FUNCTION_BLOCK FB_CalcThicknessFromXRayTransmission EXTENDS FB_Fallible IMPLEMENTS I_CalcThicknessFromXRayTransmission
VAR
    iConvertUnits : I_ConvertUnitsLREAL;
    iCalcXRayAbsorption : I_CalcXRayAbsorptionConstant;

    fbAbsorptionConstant : FB_QuantityLREALPublic(Units := '1/m');
    fbAbsorptionConstantum : FB_QuantityLREALPublic(Units := '1/um');
    fbThickness : FB_QuantityLREALPublic(Units := 'um');
END_VAR


METHOD Calculate
VAR_INPUT
    MaterialFormula : T_MaxString;
    Transmission : I_QuantityLREAL;
    Thickness : I_QuantityLREALPublic;
END_VAR

// Initialize error values
ClearError();

IF Transmission.GetError() THEN
    SetError(Msg :=
        CONCAT('Input transmission has an error: ',
        Transmission.GetErrorMsg())
    );
    Thickness.SetError(Msg := GetErrorMsg());
    RETURN;
END_IF

IF Transmission.Val <= 0.0 THEN
    SetError(Msg := 'Input transmission must be greater than 0.');
    Thickness.SetError(Msg := GetErrorMsg());
    RETURN;
END_IF

iCalcXRayAbsorption.Calculate(
    MaterialFormula := MaterialFormula,
    AbsorptionConstant := fbAbsorptionConstant
);

IF iCalcXRayAbsorption.GetError() THEN
    SetError(Msg :=
        CONCAT('Error while calculating xray absorption constant: ',
        iCalcXRayAbsorption.GetErrorMsg())
    );
    Thickness.SetError(Msg := GetErrorMsg());
    RETURN;
END_IF

IF fbAbsorptionConstant.Val <= 0.0 THEN
    SetError(Msg := 'Absorption constant must be greater than 0.');
    Thickness.SetError(Msg := GetErrorMsg());
    RETURN;
END_IF

iConvertUnits.ConvertQuantityLREAL(
    QuantityToConvert := fbAbsorptionConstant,
    DesiredUnits := fbAbsorptionConstantum.Units,
    ConvertedQuantity := fbAbsorptionConstantum
);

IF iConvertUnits.GetError() THEN
    SetError(Msg :=
        CONCAT('Error returned when attempting to convert units of absorption constant: ',
        iConvertUnits.GetErrorMsg())
    );
    Thickness.SetError(Msg := GetErrorMsg());
    RETURN;
END_IF

fbThickness.Val := LN(1.0 / Transmission.Val) / fbAbsorptionConstantum.Val;

Thickness.Copy(fbThickness);
END_METHOD


METHOD PROTECTED ClearError

SUPER^.ClearError();

fbAbsorptionConstant.ClearError();
END_METHOD


METHOD FB_init : BOOL
VAR_INPUT
    bInitRetains : BOOL; // if TRUE, the retain variables are initialized (warm start / cold start)
    bInCopyCode : BOOL;  // if TRUE, the instance afterwards gets moved into the copy code (online change)

    ConvertUnits : I_ConvertUnitsLREAL;
    CalcXRayAbsorption : I_CalcXRayAbsorptionConstant;
END_VAR

THIS^.iConvertUnits := ConvertUnits;
THIS^.iCalcXRayAbsorption := CalcXRayAbsorption;
END_METHOD


METHOD PROTECTED SetError
VAR_INPUT
    Msg : T_MaxString;
END_VAR

SUPER^.SetError(Msg := Msg);

fbAbsorptionConstant.SetError(Msg := Msg);
END_METHOD

END_FUNCTION_BLOCK

(* stored: Version 1.1.0.1
   POU FB_CalcThicknessFromXRayTransmission: Id {977af5a5-4464-419f-a60b-ad9c25dad135}, SpecialFunc None
   Method Calculate: Id {ace1d960-6880-4eb4-8c3f-5b1432b6ef56}
   Method ClearError: Id {19b39944-b5af-43fd-8404-b22953cae9a4}
   Method FB_init: Id {e1867309-abac-44c8-a3dd-7b3c96237864}
   Method SetError: Id {1b331c1b-9e69-4bdd-9311-295f846f7350} *)
